ABB RobotStudio station: CvProjekt_Pakr.rspag

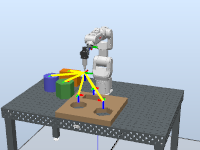
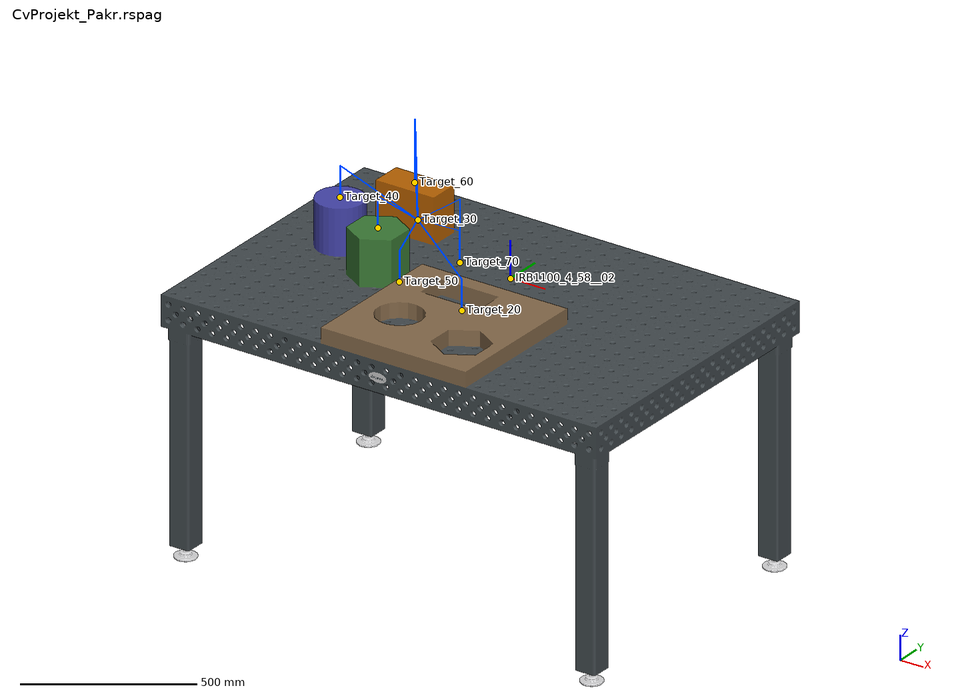
[picture v1: parts stored in the station drawn from their meshes, with robot base, taught points and paths (robot models come from the ABB library and are not in the file)]
--- station ---
Station Solution_1_Template_2 (saved by RobotStudio 21.4.9700.0)
Controller Controller2, task T_ROB1: task frame (RAPID world) sits at (0, 150, 830) mm, rotated rx 0 ry 0 rz -90 deg in the station
Controller Controller2
  mechanical unit ROB_1: IRB1100_4_58__02, 6 joints, base frame (0, 0, 0) mm
Layout (positions relative to the parent item):
  - table [part] at (-200, -500, 830) mm, size 500 x 500 x 50 mm
  - object_1 [part] at (-600, -150, 830) mm, size 200 x 100 x 150 mm
  - object_2 [part] at (-650, -150, 830) mm, size 149.5 x 149.7 x 150 mm
  - object_3 [part] at (-700, -200, 830) mm, size 155.5 x 179.5 x 150 mm
  - siegmund_1500_1000 [part], size 1500 x 1010.3 x 830 mm
  - object_11 [part] at (-200, -500, 830) mm, size 200 x 100 x 150 mm
  - object_22 [part] at (-200, -500, 830) mm, size 149.5 x 149.7 x 150 mm
  - object_33 [part] at (-200, -500, 830) mm, size 155.5 x 179.5 x 150 mm
  - IRB1100_4_58__02 [mechanism, from Robots\IRB1100_4_58__02.rslib] at (0, 150, 830) mm, rotated rx 0 ry 0 rz -90 deg; joint values [0, 0, 0, 0, 0.9076, 0] (rad or m)
  - Positioner [smart component, from Components\Positioner.rslib]
      properties: Object=object_3; Position=[-0.7 -0.2 0.83]; Orientation=[0 0 0]; Reference=Global; ReferenceObject=(none)
  - Attacher [smart component, from Components\Attacher.rslib]
      properties: Parent=MyTool_3; Flange=0; Child=object_3; Mount=false; Offset=[0 0 0]; Orientation=[0 0 0]
  - Detacher [smart component, from Components\Detacher.rslib]
      properties: Child=object_3; KeepPosition=true
  - Attacher_2 [smart component, from Components\Attacher.rslib]
      properties: Parent=MyTool_3; Flange=0; Child=object_2; Mount=false; Offset=[0 0 0]; Orientation=[0 0 0]
  - Attacher_3 [smart component, from Components\Attacher.rslib]
      properties: Parent=MyTool_3; Flange=0; Child=object_1; Mount=false; Offset=[0 0 0]; Orientation=[0 0 0]
  - Detacher_3 [smart component, from Components\Detacher.rslib]
      properties: Child=object_1; KeepPosition=true
  - Positioner_2 [smart component, from Components\Positioner.rslib]
      properties: Object=object_2; Position=[-0.65 -0.15 0.83]; Orientation=[0 0 0]; Reference=Global; ReferenceObject=(none)
  - Positioner_3 [smart component, from Components\Positioner.rslib]
      properties: Object=object_1; Position=[-0.6 -0.15 0.83]; Orientation=[0 0 0]; Reference=Global; ReferenceObject=(none)
  - MyTool_3 [mechanism, from Training Objects\myTool.rslib] at (0, -189.4, 1396.57) mm, rotated rx 180 ry 38 rz 90 deg
  - Detacher_4 [smart component, from Components\Detacher.rslib]
      properties: Child=object_2; KeepPosition=true
Attachment: MyTool_3 is attached to IRB1100_4_58__02 / Link6
Station signals: DI DI_POS_OBJ3, DI DI_POS_OBJ2, DI DI_POS_OBJ1
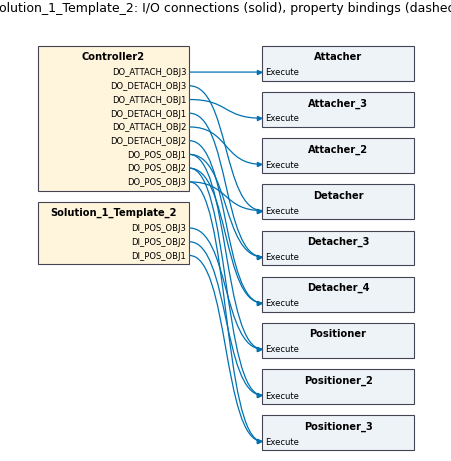
Station logic (signal -> signal, property => property):
  Controller2.DO_ATTACH_OBJ3 -> Attacher.Execute
  Controller2.DO_DETACH_OBJ3 -> Detacher.Execute
  Controller2.DO_ATTACH_OBJ1 -> Attacher_3.Execute
  Controller2.DO_DETACH_OBJ1 -> Detacher_3.Execute
  Controller2.DO_ATTACH_OBJ2 -> Attacher_2.Execute
  Solution_1_Template_2.DI_POS_OBJ3 -> Positioner.Execute
  Solution_1_Template_2.DI_POS_OBJ2 -> Positioner_2.Execute
  Solution_1_Template_2.DI_POS_OBJ1 -> Positioner_3.Execute
  Controller2.DO_DETACH_OBJ2 -> Detacher_4.Execute
  Controller2.DO_POS_OBJ1 -> Positioner.Execute
  Controller2.DO_POS_OBJ2 -> Positioner_2.Execute
  Controller2.DO_POS_OBJ3 -> Positioner_3.Execute
  Controller2.DO_POS_OBJ1 -> Detacher_3.Execute
  Controller2.DO_POS_OBJ2 -> Detacher_4.Execute
  Controller2.DO_POS_OBJ3 -> Detacher.Execute

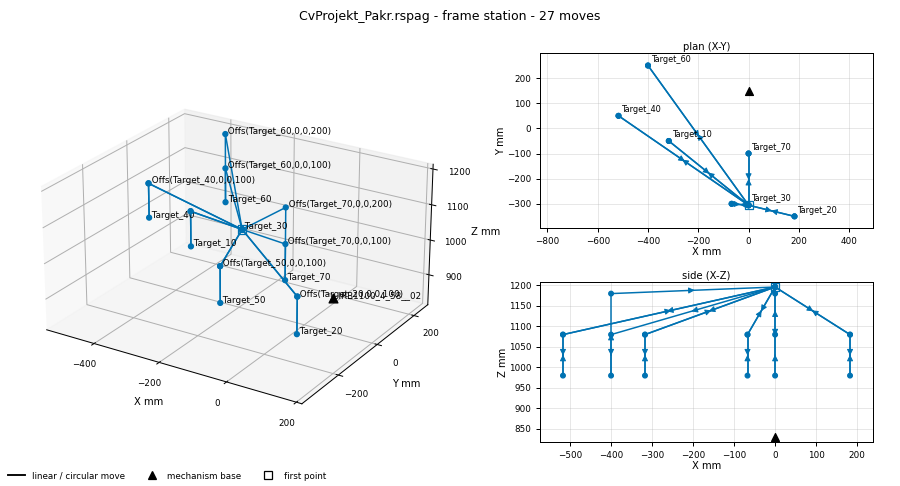
[picture p0: tool path of CvProjekt_Pakr.rspag in frame station, 27 of 27 moves have a stored position in this frame; points joined in program order, loops and branches not executed]
--- Backups/Controller2/RAPID/TASK1/PROGMOD/CalibData.modx ---
MODULE CalibData
    PERS tooldata smc_gripper:=[TRUE,[[0,0.004,197.001],[1,0,0,0]],[1,[0.207,-0.496,71.18],[1,0,0,0],0,0,0]];
    PERS tooldata Servo:=[TRUE,[[0,0,114.2],[1,0,0,0]],[0.215,[8.7,12.3,49.2],[1,0,0,0],0.00021,0.00024,0.00009]];
    PERS tooldata MyTool:=[TRUE,[[31.792631019,0,229.638935148],[0.945518576,0,0.325568154,0]],[1,[0,0,1],[1,0,0,0],0,0,0]];
ENDMODULE

--- Backups/Controller2/RAPID/TASK1/PROGMOD/Module1.modx ---
MODULE Module1
    CONST robtarget Target_30:=[[455.729,0,366.036],[0,0,1,0],[0,0,0,0],[9E+09,9E+09,9E+09,9E+09,9E+09,9E+09]];
    CONST robtarget Target_10:=[[200,-317.298,150],[0,0.707106781,0.707106781,0],[0,0,0,0],[9E+09,9E+09,9E+09,9E+09,9E+09,9E+09]];
    CONST robtarget Target_20:=[[500,182.702,150],[0,-0.707106781,0.707106781,0],[0,0,0,0],[9E+09,9E+09,9E+09,9E+09,9E+09,9E+09]];
    CONST robtarget Target_40:=[[100,-517.298,150],[0,0.707106781,0.707106781,0],[-1,-1,0,0],[9E+09,9E+09,9E+09,9E+09,9E+09,9E+09]];
    CONST robtarget Target_50:=[[450,-67.298,150],[0,0.707106781,0.707106781,0],[0,-1,1,0],[9E+09,9E+09,9E+09,9E+09,9E+09,9E+09]];
    CONST robtarget Target_60:=[[-100,-400,150],[0,0.707106781,0.707106781,0],[-2,0,-1,0],[9E+09,9E+09,9E+09,9E+09,9E+09,9E+09]];
    CONST robtarget Target_70:=[[250,0,150],[0,0.707106781,0.707106781,0],[0,-1,1,0],[9E+09,9E+09,9E+09,9E+09,9E+09,9E+09]];
!***********************************************************
    !
    ! Module:  Module1
    !
    ! Description:
    !   <Insert description here>
    !
    ! Author: Jiri
    !
    ! Version: 1.0
    !
    !***********************************************************


    !***********************************************************
    !
    ! Procedure main
    !
    !   This is the entry point of your program
    !
    !***********************************************************
    PROC main()
        PulseDO DO_POS_OBJ1;
        PulseDO DO_POS_OBJ2;
        PulseDO DO_POS_OBJ3;
        Path_10;
    ENDPROC
        PROC Path_10()

        ! OBJ 3
            !! Initial position
            MoveL Target_30,v300,fine,MyTool\WObj:=wobj0;

            !! Pick
            MoveL Offs(Target_10, 0, 0, 100), v300,fine, MyTool\WObj:=wobj0;
            MoveL Target_10,v300,fine,MyTool\WObj:=wobj0;
            WaitTime 0.1;
            PulseDO DO_ATTACH_OBJ3;    ! Pulsne signal, ktere spusti attach
            WaitTime 0.1;
            MoveL Offs(Target_10, 0, 0, 100), v300,fine, MyTool\WObj:=wobj0;

            !! Initial position
            MoveL Target_30,v300,fine,MyTool\WObj:=wobj0;

            !! Place
            MoveL Offs(Target_20, 0, 0, 100), v300,fine, MyTool\WObj:=wobj0;
            MoveL Target_20,v300,fine,MyTool\WObj:=wobj0;
            WaitTime 0.1;
            PulseDO DO_DETACH_OBJ3;    ! Pulsne signal, ktere spusti detach
            WaitTime 0.1;
            MoveL Offs(Target_20, 0, 0, 100), v300,fine, MyTool\WObj:=wobj0;

            !! Initial position
            MoveL Target_30,v300,fine,MyTool\WObj:=wobj0;


          ! OBJ 1
            !! Initial position
            MoveL Target_30,v300,fine,MyTool\WObj:=wobj0;

            !! Pick
            MoveL Offs(Target_60, 0, 0, 100), v300,fine, MyTool\WObj:=wobj0;
            MoveL Target_60,v300,fine,MyTool\WObj:=wobj0;
            WaitTime 0.1;
            PulseDO DO_ATTACH_OBJ1;
            WaitTime 0.1;
            MoveL Offs(Target_60, 0, 0, 200), v300,fine, MyTool\WObj:=wobj0;

            !! Initial position
            MoveL Target_30,v300,fine,MyTool\WObj:=wobj0;

            !! Place
            MoveL Offs(Target_70, 0, 0, 200), v300,fine, MyTool\WObj:=wobj0;
            MoveL Target_70,v300,fine,MyTool\WObj:=wobj0;
            WaitTime 0.1;
            PulseDO DO_DETACH_OBJ1;
            WaitTime 0.1;
            MoveL Offs(Target_70, 0, 0, 100), v300,fine, MyTool\WObj:=wobj0;

            !! Initial position
            MoveL Target_30,v300,fine,MyTool\WObj:=wobj0;


         ! OBJ 2
            !! Initial position
            MoveL Target_30,v300,fine,MyTool\WObj:=wobj0;

            !! Pick
            MoveL Offs(Target_40, 0, 0, 100), v300,fine, MyTool\WObj:=wobj0;
            MoveL Target_40,v300,fine,MyTool\WObj:=wobj0;
            WaitTime 0.1;
            PulseDO DO_ATTACH_OBJ2;
            WaitTime 0.1;
            MoveL Offs(Target_40, 0, 0, 100), v300,fine, MyTool\WObj:=wobj0;

            !! Initial position
            MoveL Target_30,v300,fine,MyTool\WObj:=wobj0;

            !! Place
            MoveL Offs(Target_50, 0, 0, 100), v300,fine, MyTool\WObj:=wobj0;
            MoveL Target_50,v300,fine,MyTool\WObj:=wobj0;
            WaitTime 0.1;
            PulseDO DO_DETACH_OBJ2;
            WaitTime 0.1;
            MoveL Offs(Target_50, 0, 0, 100), v300,fine, MyTool\WObj:=wobj0;

            !! Initial position
            MoveL Target_30,v300,fine,MyTool\WObj:=wobj0;
    ENDPROC
ENDMODULE

--- Backups/Controller2/SYSPAR/EIO.cfg ---
EIO:CFG_1.0:7:0::
#
EIO_SIGNAL:

      -Name "DO_ATTACH_OBJ3" -SignalType "DO" -Access "All"

      -Name "DO_DETACH_OBJ3" -SignalType "DO" -Access "All"

      -Name "DO_ATTACH_OBJ2" -SignalType "DO" -Access "All"

      -Name "DO_ATTACH_OBJ1" -SignalType "DO" -Access "All"

      -Name "DO_DETACH_OBJ2" -SignalType "DO" -Access "All"

      -Name "DO_DETACH_OBJ1" -SignalType "DO" -Access "All"

      -Name "DO_POS_OBJ1" -SignalType "DO" -Access "All"

      -Name "DO_POS_OBJ2" -SignalType "DO" -Access "All"

      -Name "DO_POS_OBJ3" -SignalType "DO" -Access "All"

#CTRL_SIGNATURE:NYgcvnZNlR/ClK2sxp65veUSRxrsIYlF/Z5I7js2hI0AwBkYYLEbisYq1nJjfEsD9620TBfCCvWqMfGO0wKylg==

--- Backups/Controller2/SYSPAR/PROC.cfg ---
PROC:CFG_1.0:7:0::

#CTRL_SIGNATURE:I+y2QaV15gWtHGM+5Z4idi3NiusZu29hLyokxM3ohwogLM8MfydOTWOtI2G6szFitByh5svEYsXD7agPogo+dQ==
